FUNCTION TryConvert_UDINT_TO_BYTE : BOOL
VAR_INPUT
	in : UDINT;
	out : REFERENCE TO BYTE;
END_VAR

IF in > DatatypeLimits.MAX_VALUE_OF_UDINT_WHICH_CAN_BE_HELD_IN_A_BYTE THEN
	RETURN;
END_IF

out := UDINT_TO_BYTE(in);
TryConvert_UDINT_TO_BYTE := TRUE;

END_FUNCTION

(* stored: Version 1.1.0.1, ProductVersion 3.1.4024.12
   POU TryConvert_UDINT_TO_BYTE: Id {02def09d-585b-4b90-ac41-96895b8eb5ae}, SpecialFunc None *)
